// TIA Portal V21 export
VAR_GLOBAL   // PLC tag table "RTD"
   "CHAMBER DRAIN TEMP" AT %IW100 : Int;
   "CHAMBER TEMP1" AT %IW102 : Int;
   "CHAMBER TEMP2" AT %IW104 : Int;
   "CHAMBER TEMP3" AT %IW106 : Int;
   "CHAMBER TEMP4" AT %IW108 : Int;
   "JACKET TEMP" AT %IW110 : Int;
END_VAR
